// TIA Portal V17 export
// export: Created 2026-04-13T11:12:44.9741801Z, ExportSetting WithDefaults, DisplayName Totally Integrated Automation Portal, DisplayVersion V17 Update 4, DisplayName TIA Portal Openness, DisplayVersion V17 Update 4, DisplayName TIA Portal Version Control Interface, DisplayVersion V17, DisplayName SINAMICS Startdrive Advanced, DisplayVersion V17, DisplayName SINAMICS Startdrive G130, G150, S120, S150, SINAMICS MV, S210, DisplayVersion V17, DisplayName SINAMICS Startdrive G110M, G120, G120C, G120D, G120P, G115D, DisplayVersion V17, DisplayName STEP 7 Professional, DisplayVersion V17 Update 4, DisplayName STEP 7 Safety, DisplayVersion V17, DisplayName WinCC Professional, DisplayVersion V17 Update 4
FUNCTION_BLOCK "PID_Compact"   // FB1130, SCL
TITLE = Compact PID_Controller with self-tuning
AUTHOR : SIMATIC
FAMILY : COMPPID
NAME : PID_Cmpt
VERSION : 2.4
// stored: IsIECCheckEnabled false, SetENOAutomatically false, UDAEnableTagReadback false
   VAR_INPUT
      Setpoint : Real;   // controller setpoint input / Sollwerteingang
      Input : Real;   // current value from process in REAL format / Istwert im REAL-Format
      Input_PER : Int;   // current value from peripheral input / Istwert im Peripherieformat
      Disturbance : Real;   // disturbance intrusion / Störaufschaltung
      ManualEnable : Bool;   // activate manual value to overwrite output value / Handwert wird zum Überschreiben des Ausgangswerts aktiviert
      ManualValue : Real;   // manual value / Handwert
      ErrorAck : Bool;   // reset error message / Löschen der Fehlermeldung
      Reset : Bool;   // reset the controller / Rücksetzen, Neustart des Reglers
      ModeActivate : Bool;   // enable mode / Modus freigeben
   END_VAR
   VAR_OUTPUT
      ScaledInput { ExternalWritable := 'False'} : Real;   // current value after scaling / Normierter Istwert
      Output { ExternalWritable := 'False'} : Real;   // output value in REAL format / Ausgangswert im REAL-Format
      Output_PER { ExternalWritable := 'False'} : Int;   // analog output value / Ausgangswert im Peripherieformat
      Output_PWM { ExternalWritable := 'False'} : Bool;   // pulse width modulated output value / Pulsweitenmodulierter Ausgangswert
      SetpointLimit_H { ExternalWritable := 'False'} : Bool;   // setpoint reached upper limit / Oberer Grenzwertmelder Sollwert
      SetpointLimit_L { ExternalWritable := 'False'} : Bool;   // setpoint reached lower limit / Unterer Grenzwertmelder Sollwert
      InputWarning_H { ExternalWritable := 'False'} : Bool;   // current value reached upper warning level / Warnung für Überschreitung der oberen Istwertwarngrenze
      InputWarning_L { ExternalWritable := 'False'} : Bool;   // current value reached lower warning level / Warnung für Unterschreitung der unteren Iswertwarngrenze
      State { ExternalWritable := 'False'} : Int;   // current mode of operation (0-Inactive, 1-SUT, 2-TIR, 3-Automatic, 4-Manual, 5-Substitute output) / Aktuelle Betriebsart (0-Inaktiv, 1-SUT, 2-TIR, 3-Automatik, 4-Hand, 5-Ersatzausgangswert)
      Error { ExternalWritable := 'False'} : Bool;   // error flag / Errorflag
      ErrorBits { ExternalWritable := 'False'} : DWord;   // error message / Fehlermeldung
   END_VAR
   VAR_IN_OUT
      Mode : Int := 4;   // mode selection / Modusanwahl
   END_VAR
   VAR
      InternalDiagnostic : DWord := 0;   // internal diagnostic and version handling / Interne Diagnose und Versionshandling
      InternalVersion { ExternalWritable := 'False'} : DWord := DW#16#02040001;   // version of controller / Version des Reglers
      InternalRTVersion : DWord := 0;   // version of runtime / Version des RunTime
      IntegralResetMode { S7_SetPoint := 'True'} : Int := 4;   // 0 smooth, 1 clear, 2 keep, 3 overwrite initial output, 4 like setpoint change / 0 glätten, 1 löschen, 2 halten, 3 Initialoutput Ablöseregelung, 4 wie Sollwertänderung
      OverwriteInitialOutputValue : Real;   // initialisation of output value for override control / Initialisierungswert des Ausgangswerts für Ablöseregelung
      RunModeByStartup { S7_SetPoint := 'True'} : Bool := true;   // activate Mode after CPU restart / Nach CPU Neustart Mode aktivieren
      LoadBackUp : Bool;   // restore last parameter set / Hochladen des Backupdatensatzes
      SetSubstituteOutput { S7_SetPoint := 'True'} : Bool := true;   // assignment of output value in State = 5 (FALSE - last valid value, TRUE - SubstituteOutput) / Belegung des Ausgangswerts bei State = 5 (FALSE - letzter gültiger Wert, TRUE - Ersatzwert SubstituteOutput)
      PhysicalUnit { ExternalWritable := 'False'; S7_SetPoint := 'True'} : Int;   // unit of measurement of the process value and setpoint / Physikalische Einheit des Ist- und Sollwerts
      PhysicalQuantity { ExternalWritable := 'False'; S7_SetPoint := 'True'} : Int;   // physical quantity of the process value and setpoint / Physikalische Größe des Ist- und Sollwerts
      ActivateRecoverMode { S7_SetPoint := 'True'} : Bool := true;   // FALSE - go to inactive by error, TRUE - activate error treatment / FALSE - gehe zu Inaktiv wenn Fehler, TRUE - Fehlerbehandlung wird aktiviert
   END_VAR
   VAR RETAIN
      Warning { ExternalWritable := 'False'} : DWord;   // warning message / Anzeige von Warnungen
      WarningInternal { ExternalWritable := 'False'} : DWord;   // warning message / Anzeige von Warnungen
   END_VAR
   VAR
      Progress { ExternalWritable := 'False'} : Real;   // progress of current phase in percent / Fortschritt der aktuellen Phase in Prozent
      CurrentSetpoint { ExternalWritable := 'False'} : Real;   // current active setpoint value / Momentan wirksamer Sollwert
      CancelTuningLevel { S7_SetPoint := 'True'} : Real := 10.0;   // cancel level for setpoint change during tuning / Abschaltschwelle für Sollwertänderung während der Selbsteinstellung
      SubstituteOutput { S7_SetPoint := 'True'} : Real;   // substitute output value in case of error / Fehlerersatzausgangswert
      Config { S7_SetPoint := 'True'} : PID_CompactConfig;   // configuration data set / Struktur mit Konfigurationsdaten
      CycleTime { S7_SetPoint := 'True'} : PID_CycleTime;   // data set for cycle time estimation / Struktur mit Variablen, zur Ermittlung der Abtastzeit
      CtrlParamsBackUp { S7_SetPoint := 'True'} : PID_CompactControlParams;   // saved parameter set / Gespeicherter Parametersatz
      PIDSelfTune { S7_SetPoint := 'True'} : PID_CompactSelfTune;   // data set for self tuning / Struktur mit Variablen für die Selbsteinstellung
      PIDCtrl { S7_SetPoint := 'True'} : PID_CompactControl;   // data for controling part / Struktur für Variablen des Reglerteils
   END_VAR
   VAR RETAIN
      Retain { S7_SetPoint := 'True'} : PID_CompactRetain;   // retain data / Struktur mit Retain-Daten
   END_VAR
BEGIN
END_FUNCTION_BLOCK
